// TwinCAT 3 PLC project main
// Title: Title
// Company: HSLU
// ProjectVersion: 2.0
// ProgramVersion: 3.1.4024.0
// libraries:
//   Tc2_Math, * (Beckhoff Automation GmbH)
//   Tc2_Standard, * (Beckhoff Automation GmbH)
//   Tc2_System, * (Beckhoff Automation GmbH)
//   Tc3_Module, * (Beckhoff Automation GmbH)
// project tree:
//   / PlcTask.TcTTO
//   POUs/ FB_EdgeDetector.TcPOU, Integrator.TcPOU, MAIN.TcPOU, PwmSignal.TcPOU, SecondOrderLag.TcPOU, SinusFunction.TcPOU, SquareSignal.TcPOU, Tiefpassfilter.TcPOU
// real-time tasks:
//   TASK PlcTask: cycle T#10ms, priority 20, ADS port 350

CONFIGURATION main
    RESOURCE PLC ON TwinCAT3
        TASK PlcTask(INTERVAL := T#10ms, PRIORITY := 20);
        PROGRAM MAIN WITH PlcTask : MAIN;
    END_RESOURCE
END_CONFIGURATION

// ---- POUs/MAIN.TcPOU
PROGRAM MAIN
VAR
END_VAR

END_PROGRAM

// ---- POUs/FB_EdgeDetector.TcPOU
FUNCTION_BLOCK FB_EdgeDetector
VAR_INPUT
	inputValue : BOOL;
	DoublePressedTime: UINT;
END_VAR
VAR_OUTPUT
	risingEdge : BOOL;
	fallingEdge : BOOL;
	DoublePressed: BOOL;
END_VAR
VAR
	inputValue_old : BOOL;
	OncePressed: BOOL := FALSE;
	DoublePressedcounter: UINT := 0;
END_VAR

risingEdge := FALSE;
fallingEdge := FALSE;
DoublePressed := FALSE;

IF inputValue <> inputValue_old THEN
	IF inputValue = TRUE THEN
		risingEdge := TRUE;
		IF OncePressed = FALSE THEN
			OncePressed := TRUE;
		ELSE
			OncePressed := FALSE;
			DoublePressed := TRUE;
			DoublePressedcounter := 0;
		END_IF
	ELSE
		fallingEdge := TRUE;
	END_IF
END_IF
inputValue_old := inputValue;
IF OncePressed = TRUE THEN
	IF DoublePressedcounter >= DoublePressedTime THEN
		OncePressed := FALSE;
		DoublePressedcounter := 0;
	ELSE
		DoublePressedcounter := DoublePressedcounter + 1;
	END_IF	
END_IF

END_FUNCTION_BLOCK

// ---- POUs/Integrator.TcPOU
FUNCTION_BLOCK Integrator
VAR_INPUT
	x : REAL;
	h : REAL;
END_VAR
VAR_OUTPUT
	y : REAL;
END_VAR
VAR
	xm : REAL;
	ym : REAL;
END_VAR

y := xm * h + ym;
ym := y;
xm := x;

END_FUNCTION_BLOCK

// ---- POUs/PwmSignal.TcPOU
FUNCTION PwmSignal : REAL
VAR_INPUT
	ymin:				REAL; 	//Minimalwert
	ymax:				REAL; 	//Maximalwert
	w:					REAL; 	//Kreisfrequenz
	yoff:				REAL; 	//yoffset
	PWM:				REAL;	//PWM 0.0 ... 1.0%
	t : 				REAL;	//Zeit
END_VAR
VAR
	tempTime:			REAL;
END_VAR

tempTime := LMOD(lr_Value:=t,lr_Arg:=(2*PI)/w)/((2*PI)/w);

IF(PWM = 1) THEN
	PwmSignal := ymax + yoff;
	RETURN;
END_IF
IF(tempTime <= (1-PWM)) THEN
	PwmSignal := ymin + yoff;
	RETURN;
ELSE
	PwmSignal := ymax + yoff;
	RETURN;
END_IF

END_FUNCTION

// ---- POUs/SecondOrderLag.TcPOU
FUNCTION_BLOCK SecondOrderLag
VAR_INPUT
	d : 	REAL;
	w : 	REAL;
	h : 	REAL;
	x : 	REAL;
END_VAR
VAR_OUTPUT
	y : 	REAL;
END_VAR
VAR
	xm : 	REAL;
	xmm : 	REAL;
	ym :	REAL;
	ymm : 	REAL;
END_VAR

y := xmm*w*w*h*h-ym*(-2+2*d*w*h)-ymm*(1-2*d*w*h+w*w*h*h);
ymm := ym;
ym := y;
xmm := xm;
xm := x;

END_FUNCTION_BLOCK

// ---- POUs/SinusFunction.TcPOU
FUNCTION SinusFunction : REAL
VAR_INPUT
	A : 	REAL; 		//Amplitude
	yoff : 	REAL;		//Offset
	w : 	REAL;		//Kreisfrequenz
	t : 	REAL;		//Zeit
END_VAR
VAR
END_VAR

SinusFunction := A * sin(w*t) + yoff;
RETURN;

END_FUNCTION

// ---- POUs/SquareSignal.TcPOU
FUNCTION SquareSignal : REAL
VAR_INPUT
	ymin:				REAL; 	//Minimalwert
	ymax:				REAL; 	//Maximalwert
	w:					REAL; 	//Kreisfrequenz
	yoff:				REAL; 	//yoffset
	t : 				REAL;	//Zeit
END_VAR
VAR
	tempTime:			REAL;
	tempVar:			INT;
END_VAR

tempTime := LMOD(lr_Value:=t,lr_Arg:=(2*PI)/w)/((2*PI)/w);

IF(tempTime >= (0.5)) THEN
	SquareSignal := ymax + yoff;
	RETURN;
ELSE
	SquareSignal := ymin + yoff;
	RETURN;
END_IF

END_FUNCTION

// ---- POUs/Tiefpassfilter.TcPOU
FUNCTION_BLOCK Tiefpassfilter
VAR_INPUT
	x : REAL;
	h : REAL;
	tau : REAL;
END_VAR
VAR_OUTPUT
	y : REAL;
END_VAR
VAR
	xm : REAL;
	ym : REAL;
END_VAR

y := (h/tau)*xm-((h/tau)-1)*ym;
ym := y;
xm := x;

END_FUNCTION_BLOCK
